FUNCTION_BLOCK CROSSCOMM_SENDER_200C0D3AE43A7966C (* Service Interface Function Block Type *)
  (* Standard: 61499-2 *)
  (* Version 0.0, 9/22/2017, bababen, nxtControl GmbH, template *)
  PACKAGE Main;
  (* Compiler Cpp nxtControl builtin 1.0 *)
  {SET_ATTRIBUTE(Runtime.FBType.ImplementingType, Runtime.System#DYNGEN_CROSSCOMM_SENDER)}
  {SET_ATTRIBUTE(Configuration.GenericFBType.InterfaceParams, Runtime.System#<InterfaceList> <EventInputs> <Event Name="CNF"> <With Var="I" /> </Event> <Event Name="INITO" /> </EventInputs> <InputVars> <VarDeclaration Name="I" Type="UINT" /> </InputVars> </InterfaceList>)}
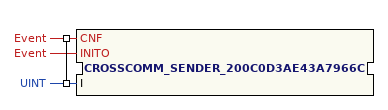
  EVENT_INPUT
    CNF WITH I;
    INITO;
  END_EVENT
  VAR_INPUT
    I : UINT;
  END_VAR
  EC_STATES
    START;
  END_STATES
END_FUNCTION_BLOCK
